{attribute 'GeneratedUsingTerminal: EL2008-0000-0018'}
{attribute addProperty VendorId "#x00000002"}
{attribute addProperty BoxType "EL2008-0000-0018"}
{attribute addProperty Description "EL2008 8Ch. Dig. Output 24V, 0.5A"}
{attribute addProperty Physics "KK"}
{attribute addProperty Id "Channel_1AT %Q*Channel_42CA91F71Channel_2AT %Q*Channel_42CA91F71Channel_3AT %Q*Channel_42CA91F71Channel_4AT %Q*Channel_42CA91F71Channel_5AT %Q*Channel_42CA91F71Channel_6AT %Q*Channel_42CA91F71Channel_7AT %Q*Channel_42CA91F71Channel_8AT %Q*Channel_42CA91F71WcStateAT %I*WcState_0B2B16F91InfoDataAT %I*InfoData_6F19DB2B2"}
{attribute addProperty CRC "3800066965"}
{attribute addProperty Size "11"}
TYPE EL2008_E2806B95 EXTENDS TcoIo.EtcSlaveTerminalBase_947E5A46 :
STRUCT
    {attribute addProperty Name "Channel_1"}
    Channel_1 : Channel_42CA91F7;
    {attribute addProperty Name "Channel_2"}
    Channel_2 : Channel_42CA91F7;
    {attribute addProperty Name "Channel_3"}
    Channel_3 : Channel_42CA91F7;
    {attribute addProperty Name "Channel_4"}
    Channel_4 : Channel_42CA91F7;
    {attribute addProperty Name "Channel_5"}
    Channel_5 : Channel_42CA91F7;
    {attribute addProperty Name "Channel_6"}
    Channel_6 : Channel_42CA91F7;
    {attribute addProperty Name "Channel_7"}
    Channel_7 : Channel_42CA91F7;
    {attribute addProperty Name "Channel_8"}
    Channel_8 : Channel_42CA91F7;
    {attribute addProperty Name "WcState"}
    WcState : TcoIo.WcState_0B2B16F9;
    {attribute addProperty Name "InfoData"}
    InfoData : TcoIo.InfoData_6F19DB2B;
END_STRUCT
END_TYPE

(* stored: Version 1.2.0.0, ProductVersion 3.1.4024.12
   DUT EL2008_E2806B95: Id {2a5d443a-b5e9-072e-1f60-fc63937c73c1} *)
